INTERFACE I_MessageData

PROPERTY DirRoot : POINTER to string(255)
SET
END_SET
END_PROPERTY

PROPERTY ErrorIndex : reference to uint
SET
END_SET
END_PROPERTY

PROPERTY FileRoot : pointer to string(255)
SET
END_SET
END_PROPERTY

PROPERTY LocalTime : pointer to DT
SET
END_SET
END_PROPERTY

PROPERTY MessageIndex : reference to uint
SET
END_SET
END_PROPERTY

PROPERTY MsgList : pointer to ARRAY[1..GVL_MSG_XTS.MAX_MESSAGE] OF st_message
SET
END_SET
END_PROPERTY

END_INTERFACE

(* stored: Version 1.1.0.1
   Itf I_MessageData: Id {48260021-0110-462c-9e4f-8e8a8dd08cb9}
   Property DirRoot: Id {c3e2af01-3ad5-48f2-9b58-2dc31653f722}
   Set Set: Id {16ce2d7f-a6bb-42cb-842d-8feb219be1e1}
   Property ErrorIndex: Id {4aef5dc9-1ad1-43e3-8e45-6861a1955285}
   Set Set: Id {fb2e462d-6fc5-4a50-88c0-d4d89d3837c8}
   Property FileRoot: Id {9ea9f99d-1a0a-40b1-a806-26df7ffa0c02}
   Set Set: Id {1c9ad8da-4bf1-4f2d-9ff3-bdb38d033368}
   Property LocalTime: Id {7870b48e-98fc-4dfd-bee8-44c6b1049760}
   Set Set: Id {e3bde52b-6469-4eeb-afad-06af73c1ff1d}
   Property MessageIndex: Id {4f8a49dd-111c-4c4b-9a99-7ea550ef9f5b}
   Set Set: Id {42ba1132-3f92-4da6-bf8d-a085ce303ea1}
   Property MsgList: Id {1e606063-8de7-442d-900c-7480207e6636}
   Set Set: Id {fde3c6ed-601a-480d-9091-c1f7c65326cc} *)
